VAR_GLOBAL
	
	iq_stM2SelectorA	:	ST_M2SelectorIO;
	iq_stM2SelectorB	:	ST_M2SelectorIO;

	iq_stM3SelectorA	:	ST_M3SelectorIO;
	iq_stM3SelectorB	:	ST_M3SelectorIO;

	i_iFscEB1Ch0AI	AT	%I*	:	INT;
	i_iFscEB1Ch1AI	AT	%I*	:	INT;
	i_iFscEB1Ch2AI	AT	%I*	:	INT;
	i_iFscEB1Ch3AI	AT	%I*	:	INT;

END_VAR

(* stored: Version 1.1.0.1, ProductVersion 3.1.4020.6
   GVL GVL_IO: Id {72fbb778-259d-42b9-8ccf-d5ffd47335bc} *)
